(* Logix 5000 project; controller LeakTestAuto vendor 1 type 14 code 226 rev 37.11; software revision 37.01; part 9 of 12 *)
(* tags used below, declared in another part *)
   AOI_Barcode_Comms : AOI_CommStatus;
   AOI_CTS1_Comms : AOI_CommStatus;
   AOI_CTS2_Comms : AOI_CommStatus;
   AOI_RFID_Comms : AOI_CommStatus;
   AOI_RFID_LoadingNest_Comms : AOI_CommStatus;
   AOI_Robot_Comms : AOI_CommStatus;
   BarcodeScanner : udt_OutputStructure;
   Conveyor : udt_OutputStructure;
   Conveyor_Seq : udt_SequenceStructure_X64;
   ConveyorCleatSensorFault : BOOL;
   FailCount : COUNTER;
   HMI_OP220_ClearProcessFaultCounts_IND : BOOL;
   HMI_OP220_ClearProcessFaultCounts_PB : BOOL;
   LastFaults : DINT[2];
   LeakTester1 : udt_OutputStructure;
   LeakTester2 : udt_OutputStructure;
   Nest1Cylinder : udt_OutputStructure;
   Nest2Cylinder : udt_OutputStructure;
   OP220 : udt_Mode;
   OP220_Disable3510 : BOOL;
   OP220_Fault_Counter : COUNTER;
   OP220_Fault_Counter_ONS : BOOL;
   OP220_Fault_Number : DINT;
   OP220_Fault_Reset_ONS : BOOL;
   OP220_FaultCounter_Reset_ONS : BOOL;
   OP220_LeakTest : udt_ProcessFault;
   OP220_ProcessFaultsONS : DINT;
   OP220_Seq : udt_SequenceStructure_X64;
   RFID_Comp : AOI_RFIDCompare;
   RFID_DiagData : DINT[4];
   RFID_ExpectedFixtureVal : SINT[5,12];
   RFID_LoadingNestDiagData : DINT[4];
   RFID_LoadingNestReceiveBuffer : SINT[8000];
   RFID_LoadingNestSendBuffer : SINT[8000];
   RFID_PortOffset : DINT;
   RFID_ReceiveBuffer : SINT[8000];
   RFID_RWHAllPort : RWH_CMD;
   RFID_RWHLoadingNest : RWH_CMD;
   RFID_SendBuffer : SINT[8000];
   RFID_TagStatus : BOOL[32];
   RFIDLoadingNestScanner : udt_OutputStructure;
   RFIDScanner : udt_OutputStructure;
   Robot : udt_OutputStructure;
   RobotGripper : udt_OutputStructure;
   RobotInputs : udt_EpsonInputs;
   TON_Cylinder1DownTimeout : TIMER;
   TON_Cylinder1UpTimeout : TIMER;
   TON_Cylinder2DownTimeout : TIMER;
   TON_Cylinder2UpTimeout : TIMER;
   TON_FailChute : TIMER[10];
   TON_Nest2CylinderTimer : TIMER;
   I_OP220_N3_MAIN_AIR_OK : ALIAS FOR Local:3:I.Pt07.Data;
   I_OP220_N3_NEST2_EXTEND : ALIAS FOR Local:3:I.Pt06.Data;
   I_OP220_N3_NEST2_HOME : ALIAS FOR Local:3:I.Pt05.Data;
   I_OP220_N3_REJECT_BIN_OK : ALIAS FOR Local:3:I.Pt09.Data;
   I_OP220_N4_DC_OK : ALIAS FOR Local:4:I.Pt01.Data;
   I_OP220_N4_DC_OK_PS2 : ALIAS FOR Local:4:I.Pt04.Data;
   James_Dint : DINT;   // James Test Word
   O_OP220_N5_EN_NEST2_EXT : ALIAS FOR Local:5:O.Pt07.Data;
   O_OP220_N5_EN_NEST2_HOME : ALIAS FOR Local:5:O.Pt08.Data;
   OP220_ConsumedFromMain : DINT[50];
   OP220_EStopTest_DCS : DCI_STOP;
   PLC : AOI_PLC;
   ShiftChange : BOOL;
(* MainProgram, continued *)

ROUTINE R61_Nest2Cylinder   (* ladder *)
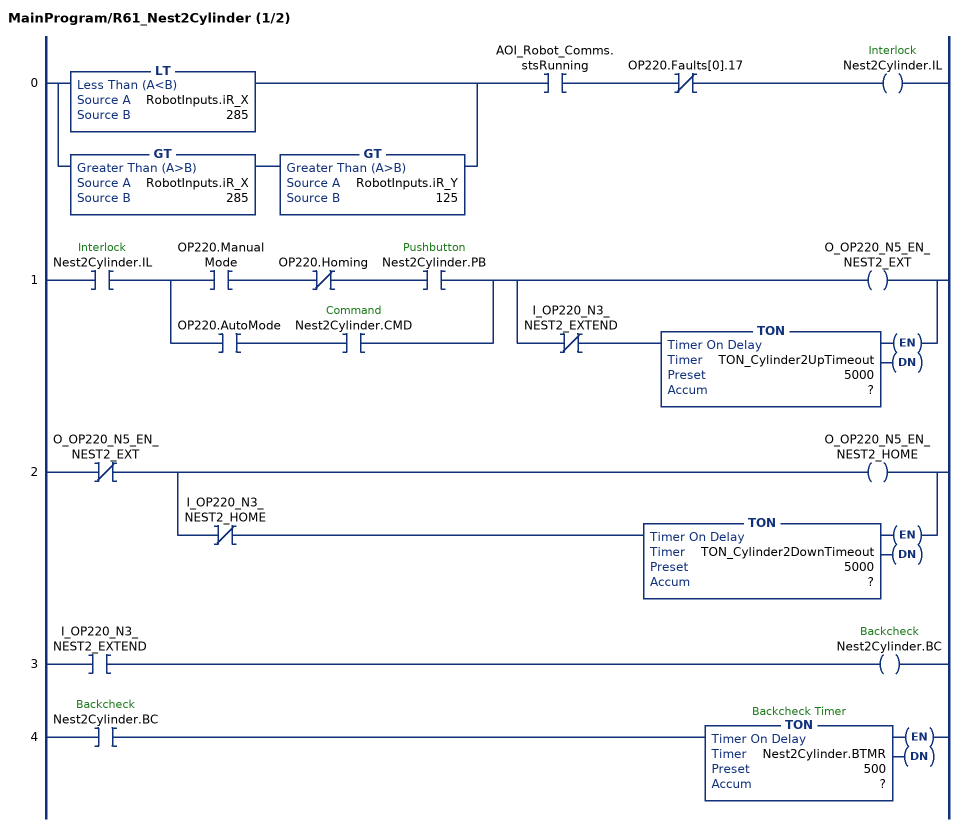
   0: [LT(RobotInputs.iR_X,285) ,GT(RobotInputs.iR_X,285) GT(RobotInputs.iR_Y,125) ]XIC(AOI_Robot_Comms.stsRunning)XIO(OP220.Faults[0].17)OTE(Nest2Cylinder.IL);
   1: XIC(Nest2Cylinder.IL)[XIC(OP220.ManualMode) XIO(OP220.Homing) XIC(Nest2Cylinder.PB) ,XIC(OP220.AutoMode) XIC(Nest2Cylinder.CMD) ][OTE(O_OP220_N5_EN_NEST2_EXT) ,XIO(I_OP220_N3_NEST2_EXTEND) TON(TON_Cylinder2UpTimeout,?,?) ];
   2: XIO(O_OP220_N5_EN_NEST2_EXT)[OTE(O_OP220_N5_EN_NEST2_HOME) ,XIO(I_OP220_N3_NEST2_HOME) TON(TON_Cylinder2DownTimeout,?,?) ];
   3: XIC(I_OP220_N3_NEST2_EXTEND)OTE(Nest2Cylinder.BC);
   4: XIC(Nest2Cylinder.BC)TON(Nest2Cylinder.BTMR,?,?);
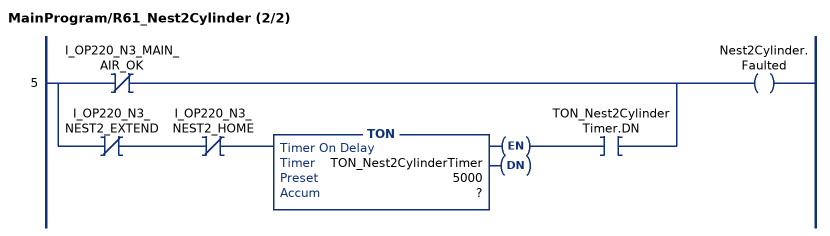
   5: [XIO(I_OP220_N3_MAIN_AIR_OK) ,XIO(I_OP220_N3_NEST2_EXTEND) XIO(I_OP220_N3_NEST2_HOME) TON(TON_Nest2CylinderTimer,?,?) XIC(TON_Nest2CylinderTimer.DN) ]OTE(Nest2Cylinder.Faulted);
END_ROUTINE

ROUTINE R70_RFID   (* ladder *)
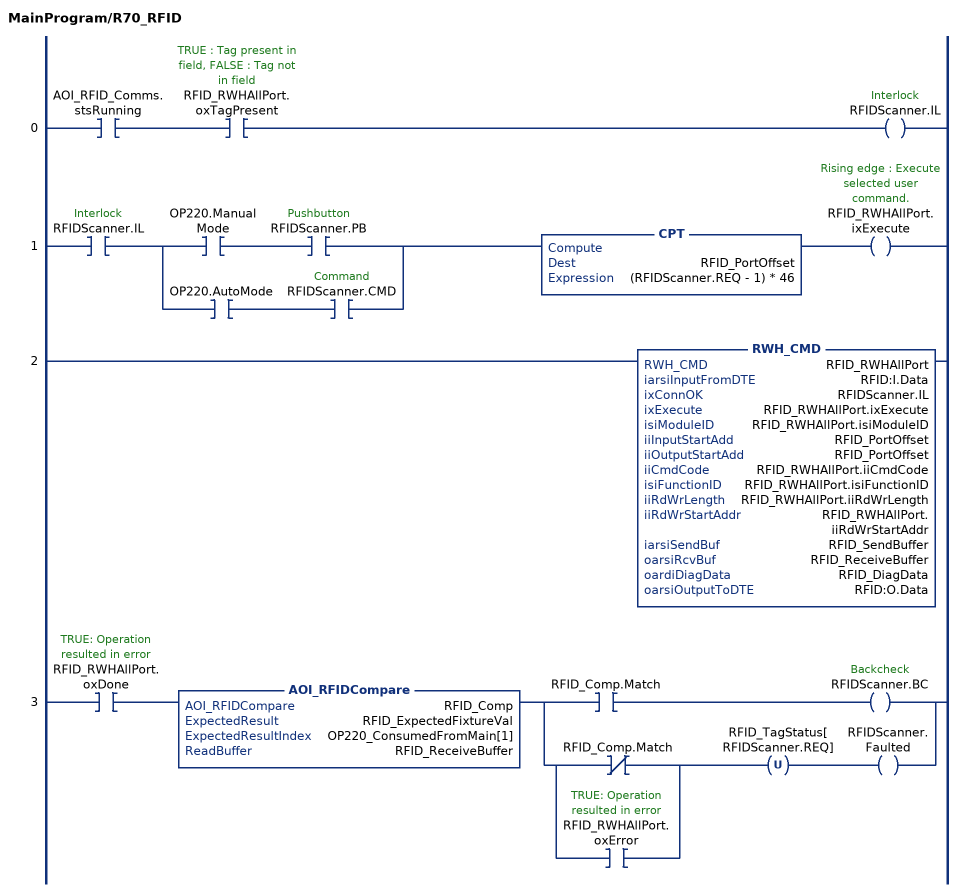
   0: XIC(AOI_RFID_Comms.stsRunning)XIC(RFID_RWHAllPort.oxTagPresent)OTE(RFIDScanner.IL);
   1: XIC(RFIDScanner.IL)[XIC(OP220.ManualMode) XIC(RFIDScanner.PB) ,XIC(OP220.AutoMode) XIC(RFIDScanner.CMD) ]CPT(RFID_PortOffset,(RFIDScanner.REQ - 1) * 46)OTE(RFID_RWHAllPort.ixExecute);
   2: RWH_CMD(RFID_RWHAllPort,RFID:I.Data,RFIDScanner.IL,RFID_RWHAllPort.ixExecute,RFID_RWHAllPort.isiModuleID,RFID_PortOffset,RFID_PortOffset,RFID_RWHAllPort.iiCmdCode,RFID_RWHAllPort.isiFunctionID,RFID_RWHAllPort.iiRdWrLength,RFID_RWHAllPort.iiRdWrStartAddr,RFID_SendBuffer,RFID_ReceiveBuffer,RFID_DiagData,RFID:O.Data);
   3: XIC(RFID_RWHAllPort.oxDone)AOI_RFIDCompare(RFID_Comp,RFID_ExpectedFixtureVal,OP220_ConsumedFromMain[1],RFID_ReceiveBuffer)[XIC(RFID_Comp.Match) OTE(RFIDScanner.BC) ,[XIO(RFID_Comp.Match) ,XIC(RFID_RWHAllPort.oxError) ] OTU(RFID_TagStatus[RFIDScanner.REQ]) OTE(RFIDScanner.Faulted) ];
END_ROUTINE

ROUTINE R71_RFID_LoadingNest   (* ladder *)
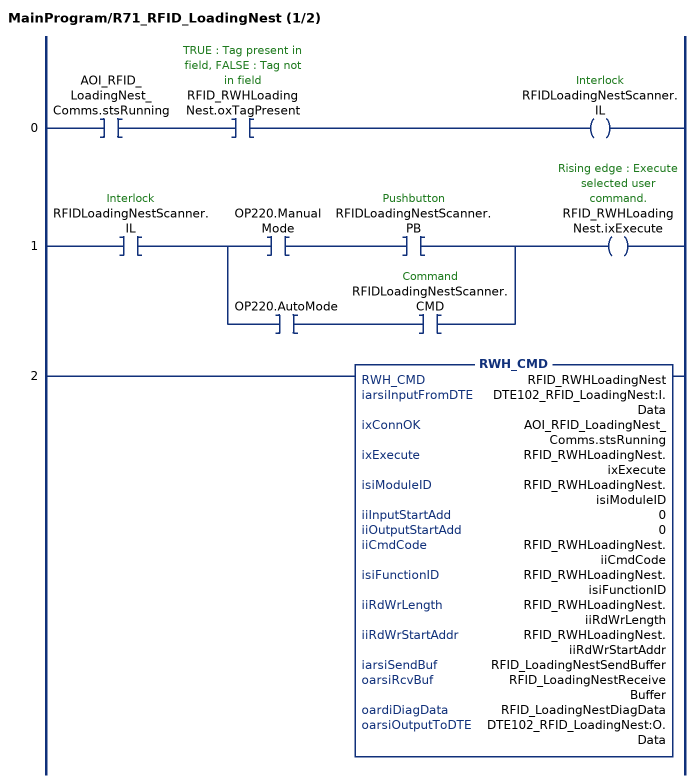
   0: XIC(AOI_RFID_LoadingNest_Comms.stsRunning)XIC(RFID_RWHLoadingNest.oxTagPresent)OTE(RFIDLoadingNestScanner.IL);
   1: XIC(RFIDLoadingNestScanner.IL)[XIC(OP220.ManualMode) XIC(RFIDLoadingNestScanner.PB) ,XIC(OP220.AutoMode) XIC(RFIDLoadingNestScanner.CMD) ]OTE(RFID_RWHLoadingNest.ixExecute);
   2: RWH_CMD(RFID_RWHLoadingNest,DTE102_RFID_LoadingNest:I.Data,AOI_RFID_LoadingNest_Comms.stsRunning,RFID_RWHLoadingNest.ixExecute,RFID_RWHLoadingNest.isiModuleID,0,0,RFID_RWHLoadingNest.iiCmdCode,RFID_RWHLoadingNest.isiFunctionID,RFID_RWHLoadingNest.iiRdWrLength,RFID_RWHLoadingNest.iiRdWrStartAddr,RFID_LoadingNestSendBuffer,RFID_LoadingNestReceiveBuffer,RFID_LoadingNestDiagData,DTE102_RFID_LoadingNest:O.Data);
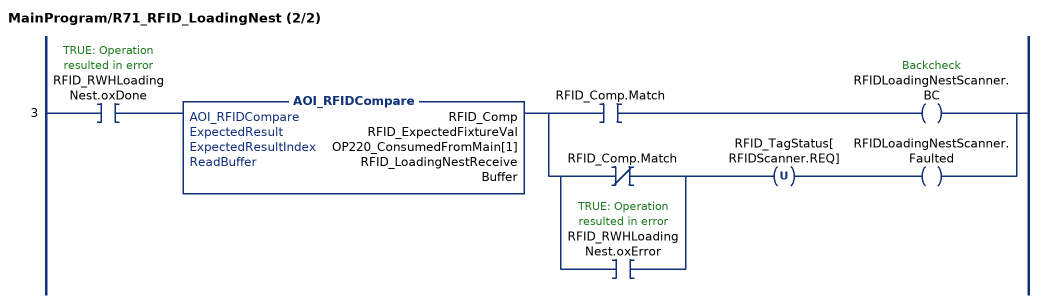
   3: XIC(RFID_RWHLoadingNest.oxDone)AOI_RFIDCompare(RFID_Comp,RFID_ExpectedFixtureVal,OP220_ConsumedFromMain[1],RFID_LoadingNestReceiveBuffer)[XIC(RFID_Comp.Match) OTE(RFIDLoadingNestScanner.BC) ,[XIO(RFID_Comp.Match) ,XIC(RFID_RWHLoadingNest.oxError) ] OTU(RFID_TagStatus[RFIDScanner.REQ]) OTE(RFIDLoadingNestScanner.Faulted) ];
END_ROUTINE

ROUTINE R89_3_5_10_Alarms   (* ladder *)
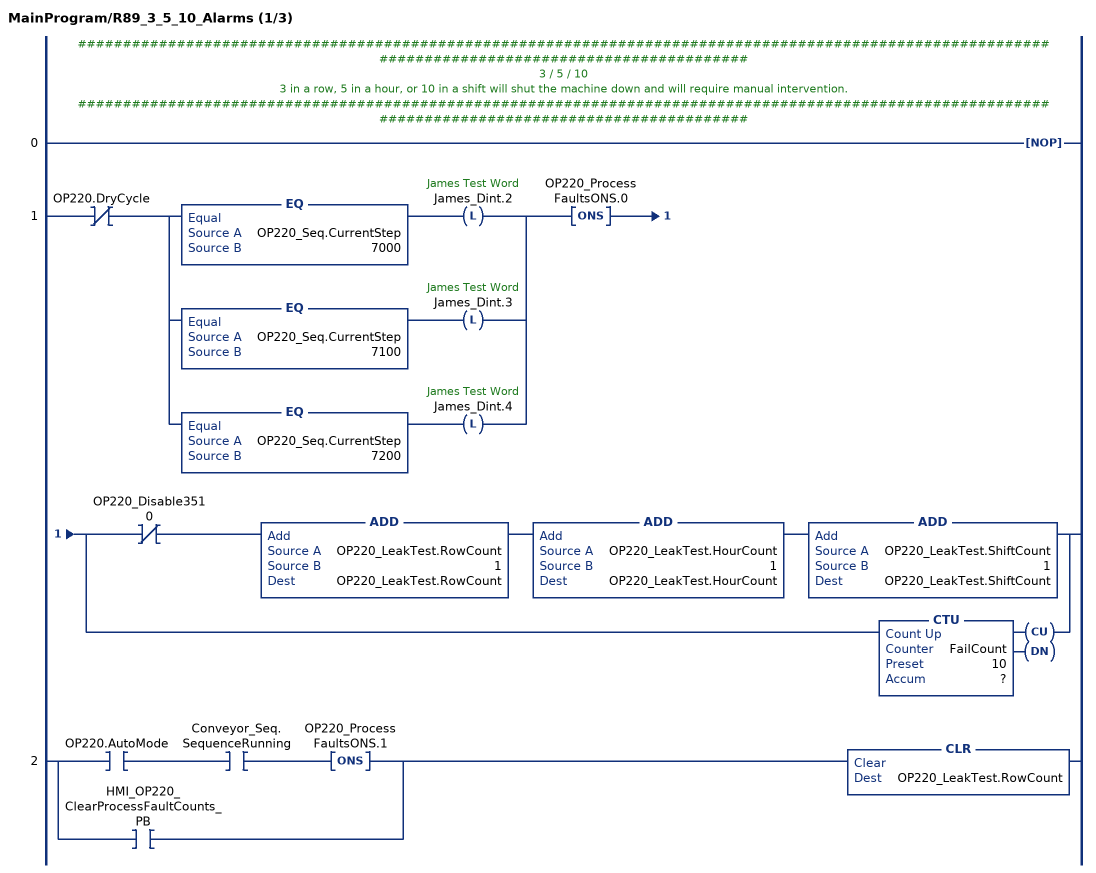
   // #####################################################################################################################################################
   // 3 / 5 / 10
   // 	3 in a row, 5 in a hour, or 10 in a shift will shut the machine down and will require manual intervention.
   // #####################################################################################################################################################
   0: NOP();
   1: XIO(OP220.DryCycle)[EQ(OP220_Seq.CurrentStep,7000) OTL(James_Dint.2) ,EQ(OP220_Seq.CurrentStep,7100) OTL(James_Dint.3) ,EQ(OP220_Seq.CurrentStep,7200) OTL(James_Dint.4) ]ONS(OP220_ProcessFaultsONS.0)[XIO(OP220_Disable3510) ADD(OP220_LeakTest.RowCount,1,OP220_LeakTest.RowCount) ADD(OP220_LeakTest.HourCount,1,OP220_LeakTest.HourCount) ADD(OP220_LeakTest.ShiftCount,1,OP220_LeakTest.ShiftCount) ,CTU(FailCount,?,?) ];
   2: [XIC(OP220.AutoMode) XIC(Conveyor_Seq.SequenceRunning) ONS(OP220_ProcessFaultsONS.1) ,XIC(HMI_OP220_ClearProcessFaultCounts_PB) ]CLR(OP220_LeakTest.RowCount);
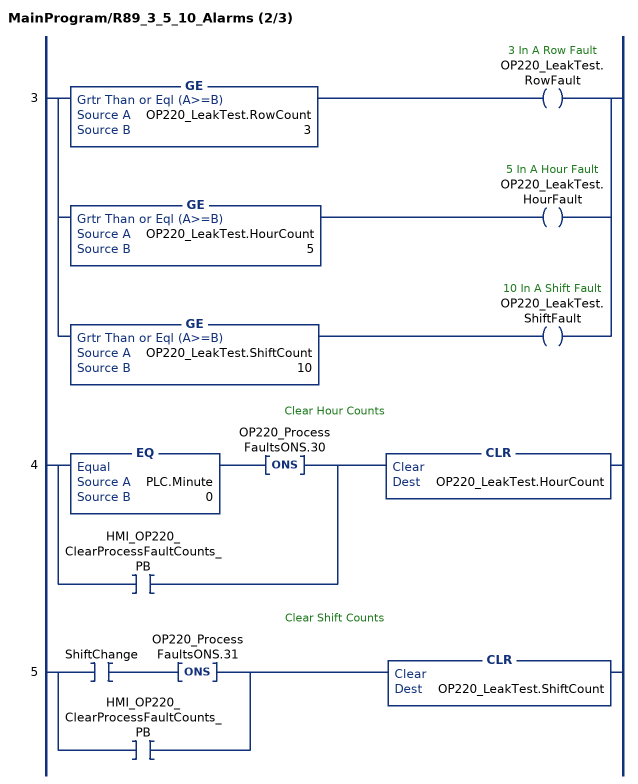
   3: [GE(OP220_LeakTest.RowCount,3) OTE(OP220_LeakTest.RowFault) ,GE(OP220_LeakTest.HourCount,5) OTE(OP220_LeakTest.HourFault) ,GE(OP220_LeakTest.ShiftCount,10) OTE(OP220_LeakTest.ShiftFault) ];
   // Clear Hour Counts
   4: [EQ(PLC.Minute,0) ONS(OP220_ProcessFaultsONS.30) ,XIC(HMI_OP220_ClearProcessFaultCounts_PB) ]CLR(OP220_LeakTest.HourCount);
   // Clear Shift Counts
   5: [XIC(ShiftChange) ONS(OP220_ProcessFaultsONS.31) ,XIC(HMI_OP220_ClearProcessFaultCounts_PB) ]CLR(OP220_LeakTest.ShiftCount);
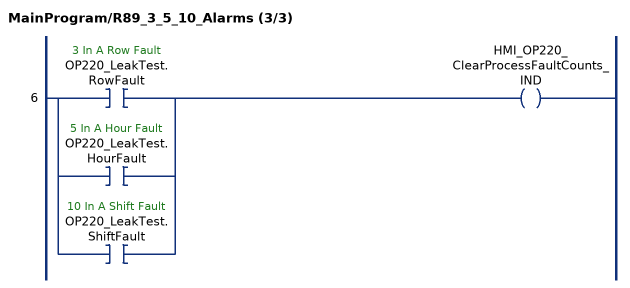
   6: [XIC(OP220_LeakTest.RowFault) ,XIC(OP220_LeakTest.HourFault) ,XIC(OP220_LeakTest.ShiftFault) ]OTE(HMI_OP220_ClearProcessFaultCounts_IND);
END_ROUTINE

ROUTINE R90_Faults   (* ladder *)
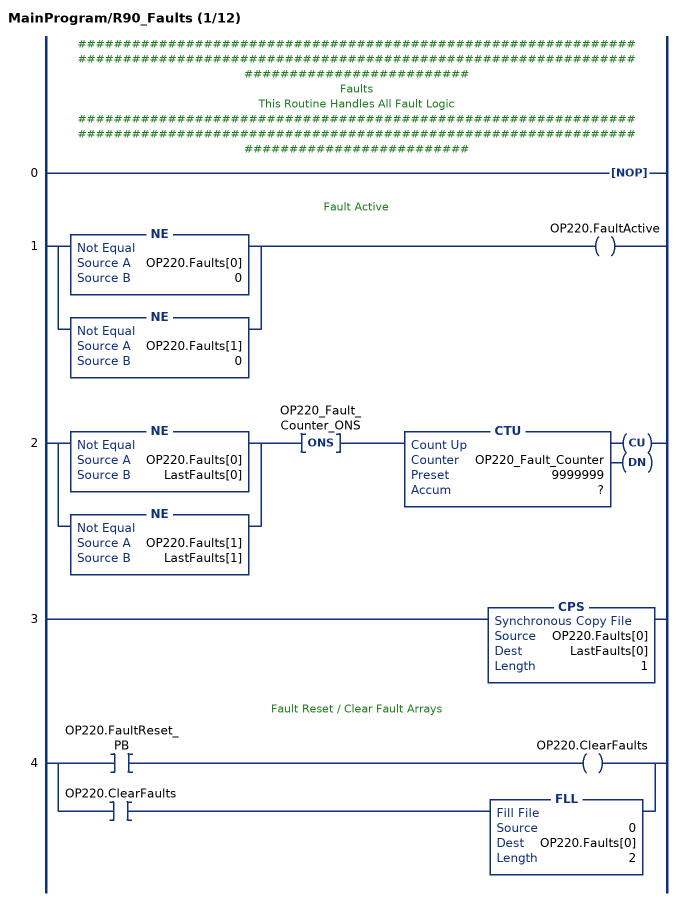
   // #####################################################################################################################################################
   // Faults
   // This Routine Handles All Fault Logic
   // #####################################################################################################################################################
   0: NOP();
   // Fault Active
   1: [NE(OP220.Faults[0],0) ,NE(OP220.Faults[1],0) ]OTE(OP220.FaultActive);
   2: [NE(OP220.Faults[0],LastFaults[0]) ,NE(OP220.Faults[1],LastFaults[1]) ]ONS(OP220_Fault_Counter_ONS)CTU(OP220_Fault_Counter,?,?);
   3: CPS(OP220.Faults[0],LastFaults[0],1);
   // Fault Reset / Clear Fault Arrays
   4: [XIC(OP220.FaultReset_PB) OTE(OP220.ClearFaults) ,XIC(OP220.ClearFaults) FLL(0,OP220.Faults[0],2) ];
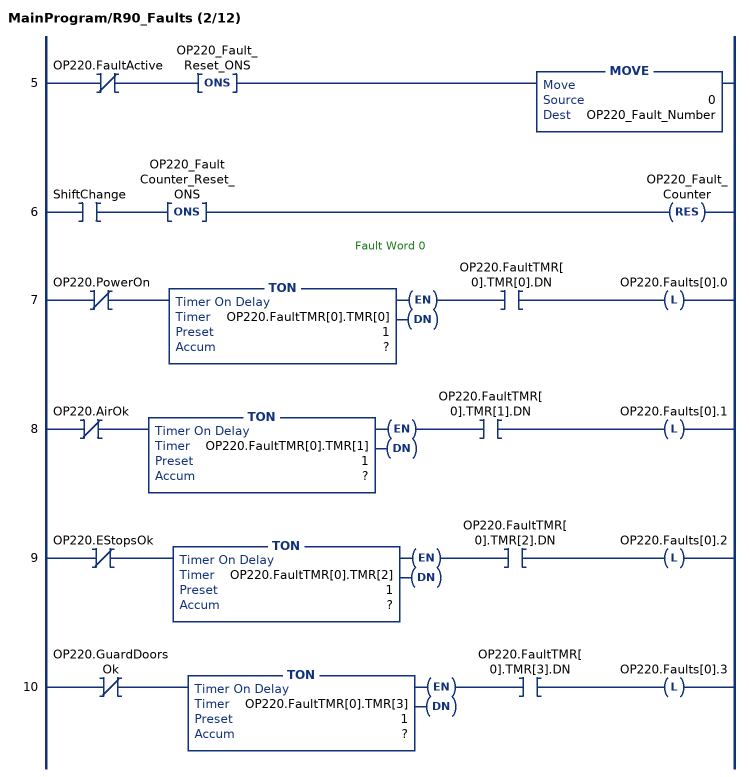
   5: XIO(OP220.FaultActive)ONS(OP220_Fault_Reset_ONS)MOVE(0,OP220_Fault_Number);
   6: XIC(ShiftChange)ONS(OP220_FaultCounter_Reset_ONS)RES(OP220_Fault_Counter);
   // Fault Word 0
   7: XIO(OP220.PowerOn)TON(OP220.FaultTMR[0].TMR[0],?,?)XIC(OP220.FaultTMR[0].TMR[0].DN)OTL(OP220.Faults[0].0);
   8: XIO(OP220.AirOk)TON(OP220.FaultTMR[0].TMR[1],?,?)XIC(OP220.FaultTMR[0].TMR[1].DN)OTL(OP220.Faults[0].1);
   9: XIO(OP220.EStopsOk)TON(OP220.FaultTMR[0].TMR[2],?,?)XIC(OP220.FaultTMR[0].TMR[2].DN)OTL(OP220.Faults[0].2);
   10: XIO(OP220.GuardDoorsOk)TON(OP220.FaultTMR[0].TMR[3],?,?)XIC(OP220.FaultTMR[0].TMR[3].DN)OTL(OP220.Faults[0].3);
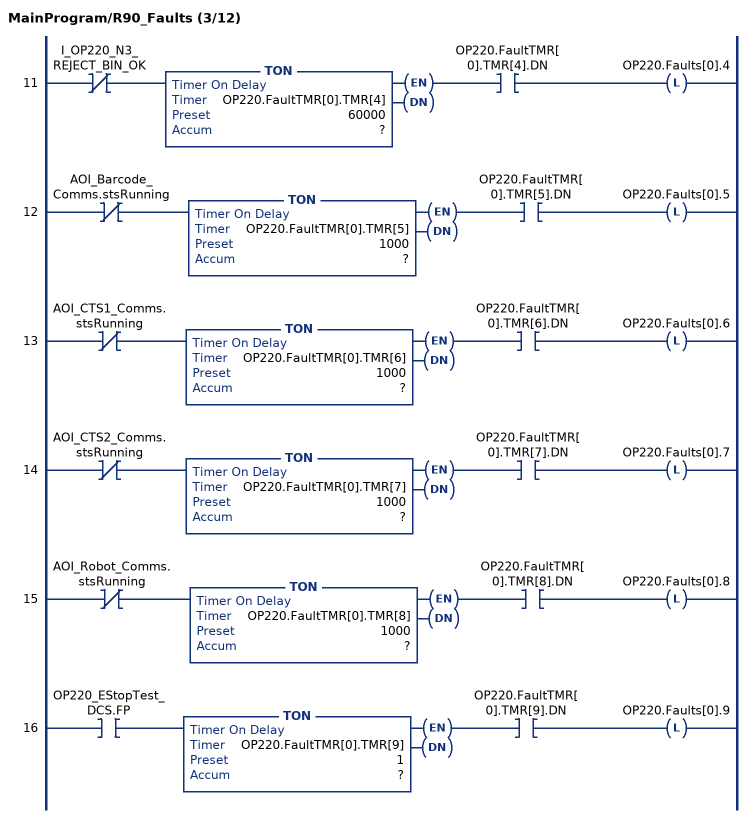
   11: XIO(I_OP220_N3_REJECT_BIN_OK)TON(OP220.FaultTMR[0].TMR[4],?,?)XIC(OP220.FaultTMR[0].TMR[4].DN)OTL(OP220.Faults[0].4);
   12: XIO(AOI_Barcode_Comms.stsRunning)TON(OP220.FaultTMR[0].TMR[5],?,?)XIC(OP220.FaultTMR[0].TMR[5].DN)OTL(OP220.Faults[0].5);
   13: XIO(AOI_CTS1_Comms.stsRunning)TON(OP220.FaultTMR[0].TMR[6],?,?)XIC(OP220.FaultTMR[0].TMR[6].DN)OTL(OP220.Faults[0].6);
   14: XIO(AOI_CTS2_Comms.stsRunning)TON(OP220.FaultTMR[0].TMR[7],?,?)XIC(OP220.FaultTMR[0].TMR[7].DN)OTL(OP220.Faults[0].7);
   15: XIO(AOI_Robot_Comms.stsRunning)TON(OP220.FaultTMR[0].TMR[8],?,?)XIC(OP220.FaultTMR[0].TMR[8].DN)OTL(OP220.Faults[0].8);
   16: XIC(OP220_EStopTest_DCS.FP)TON(OP220.FaultTMR[0].TMR[9],?,?)XIC(OP220.FaultTMR[0].TMR[9].DN)OTL(OP220.Faults[0].9);
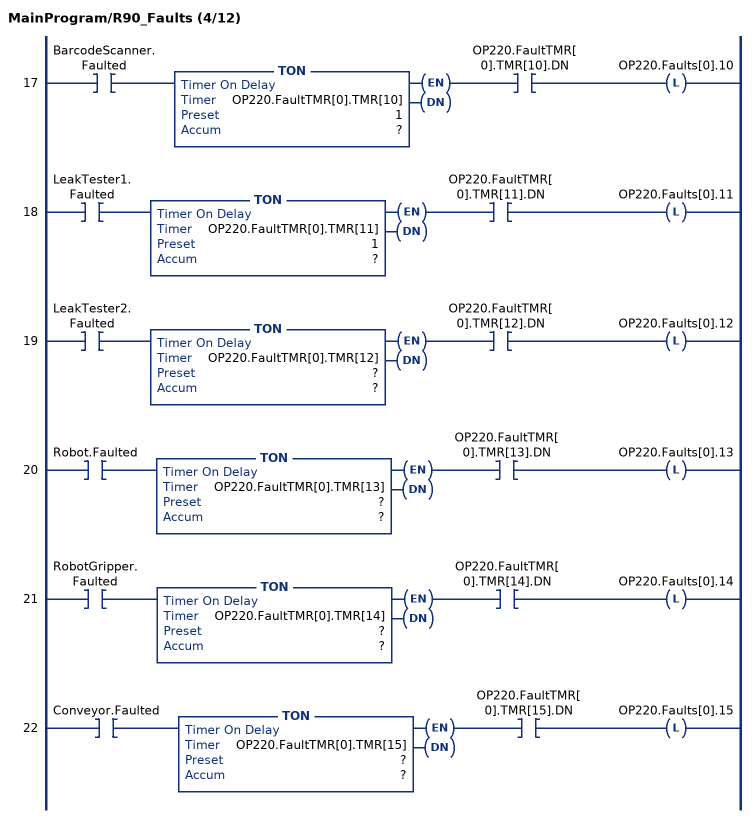
   17: XIC(BarcodeScanner.Faulted)TON(OP220.FaultTMR[0].TMR[10],?,?)XIC(OP220.FaultTMR[0].TMR[10].DN)OTL(OP220.Faults[0].10);
   18: XIC(LeakTester1.Faulted)TON(OP220.FaultTMR[0].TMR[11],?,?)XIC(OP220.FaultTMR[0].TMR[11].DN)OTL(OP220.Faults[0].11);
   19: XIC(LeakTester2.Faulted)TON(OP220.FaultTMR[0].TMR[12],?,?)XIC(OP220.FaultTMR[0].TMR[12].DN)OTL(OP220.Faults[0].12);
   20: XIC(Robot.Faulted)TON(OP220.FaultTMR[0].TMR[13],?,?)XIC(OP220.FaultTMR[0].TMR[13].DN)OTL(OP220.Faults[0].13);
   21: XIC(RobotGripper.Faulted)TON(OP220.FaultTMR[0].TMR[14],?,?)XIC(OP220.FaultTMR[0].TMR[14].DN)OTL(OP220.Faults[0].14);
   22: XIC(Conveyor.Faulted)TON(OP220.FaultTMR[0].TMR[15],?,?)XIC(OP220.FaultTMR[0].TMR[15].DN)OTL(OP220.Faults[0].15);
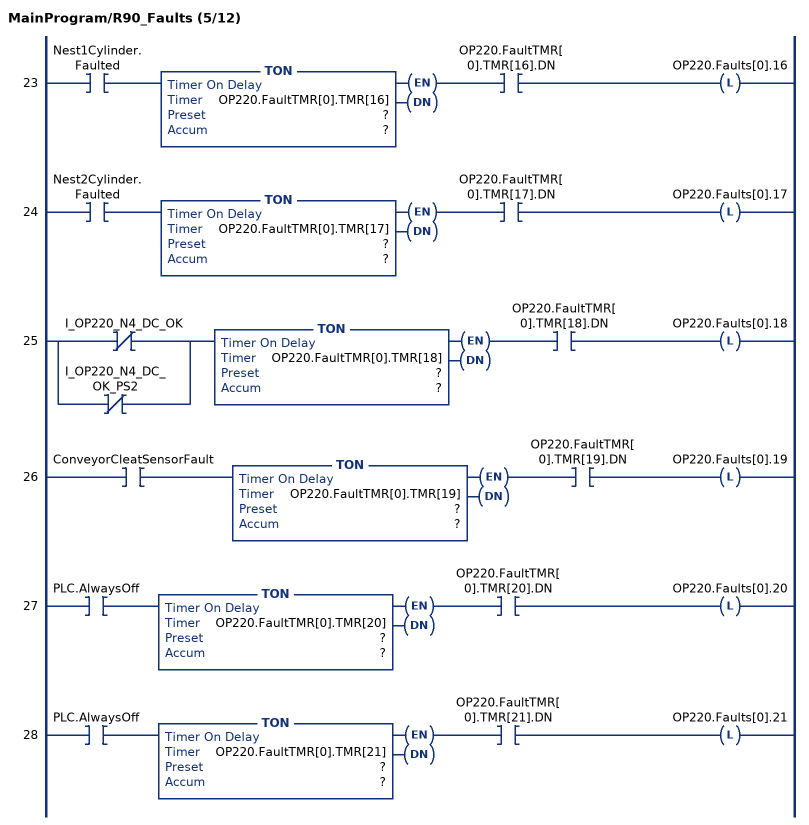
   23: XIC(Nest1Cylinder.Faulted)TON(OP220.FaultTMR[0].TMR[16],?,?)XIC(OP220.FaultTMR[0].TMR[16].DN)OTL(OP220.Faults[0].16);
   24: XIC(Nest2Cylinder.Faulted)TON(OP220.FaultTMR[0].TMR[17],?,?)XIC(OP220.FaultTMR[0].TMR[17].DN)OTL(OP220.Faults[0].17);
   25: [XIO(I_OP220_N4_DC_OK) ,XIO(I_OP220_N4_DC_OK_PS2) ]TON(OP220.FaultTMR[0].TMR[18],?,?)XIC(OP220.FaultTMR[0].TMR[18].DN)OTL(OP220.Faults[0].18);
   26: XIC(ConveyorCleatSensorFault)TON(OP220.FaultTMR[0].TMR[19],?,?)XIC(OP220.FaultTMR[0].TMR[19].DN)OTL(OP220.Faults[0].19);
   27: XIC(PLC.AlwaysOff)TON(OP220.FaultTMR[0].TMR[20],?,?)XIC(OP220.FaultTMR[0].TMR[20].DN)OTL(OP220.Faults[0].20);
   28: XIC(PLC.AlwaysOff)TON(OP220.FaultTMR[0].TMR[21],?,?)XIC(OP220.FaultTMR[0].TMR[21].DN)OTL(OP220.Faults[0].21);
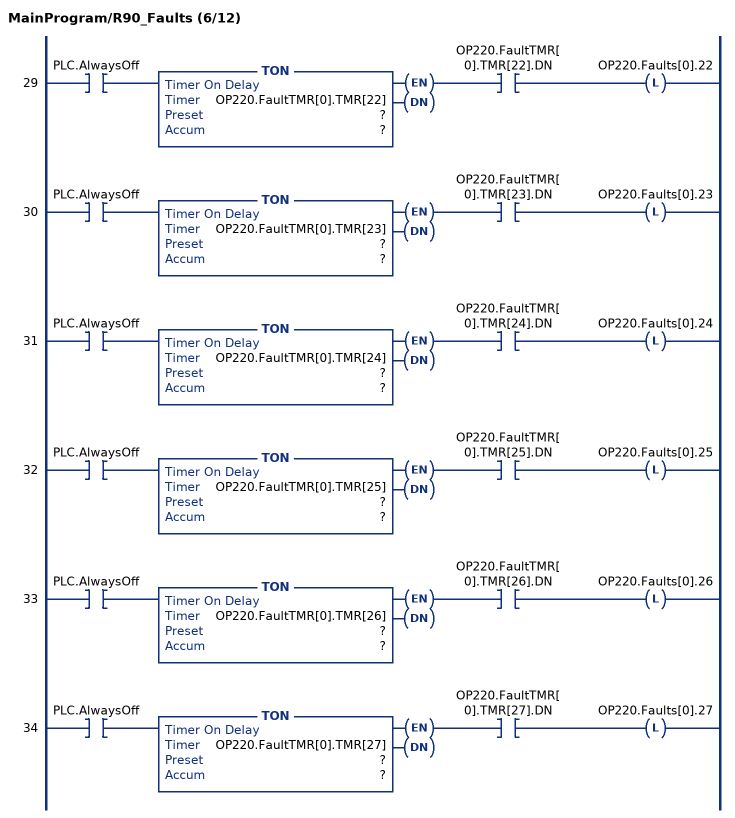
   29: XIC(PLC.AlwaysOff)TON(OP220.FaultTMR[0].TMR[22],?,?)XIC(OP220.FaultTMR[0].TMR[22].DN)OTL(OP220.Faults[0].22);
   30: XIC(PLC.AlwaysOff)TON(OP220.FaultTMR[0].TMR[23],?,?)XIC(OP220.FaultTMR[0].TMR[23].DN)OTL(OP220.Faults[0].23);
   31: XIC(PLC.AlwaysOff)TON(OP220.FaultTMR[0].TMR[24],?,?)XIC(OP220.FaultTMR[0].TMR[24].DN)OTL(OP220.Faults[0].24);
   32: XIC(PLC.AlwaysOff)TON(OP220.FaultTMR[0].TMR[25],?,?)XIC(OP220.FaultTMR[0].TMR[25].DN)OTL(OP220.Faults[0].25);
   33: XIC(PLC.AlwaysOff)TON(OP220.FaultTMR[0].TMR[26],?,?)XIC(OP220.FaultTMR[0].TMR[26].DN)OTL(OP220.Faults[0].26);
   34: XIC(PLC.AlwaysOff)TON(OP220.FaultTMR[0].TMR[27],?,?)XIC(OP220.FaultTMR[0].TMR[27].DN)OTL(OP220.Faults[0].27);
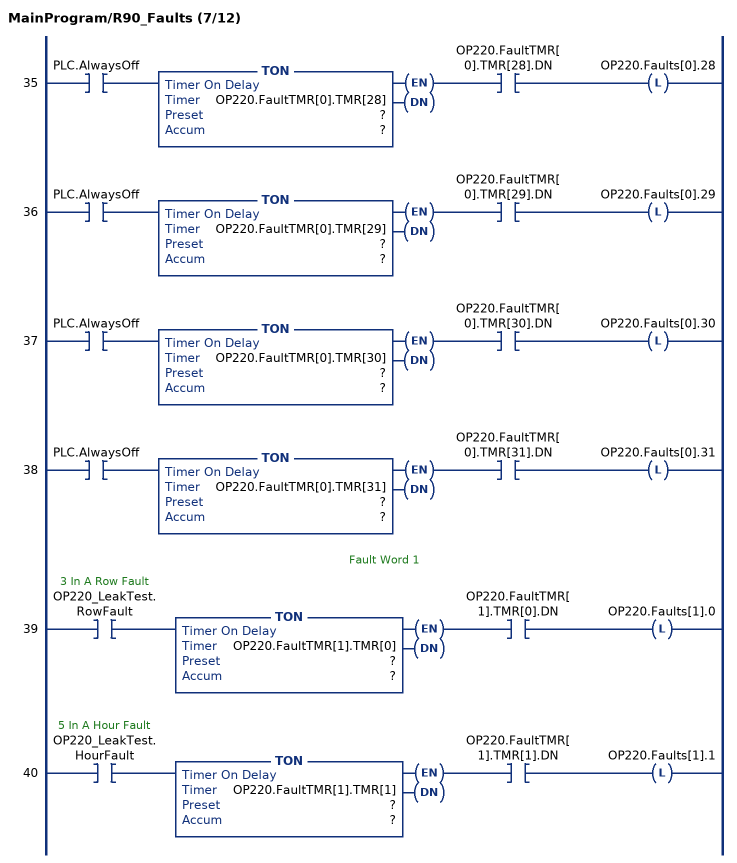
   35: XIC(PLC.AlwaysOff)TON(OP220.FaultTMR[0].TMR[28],?,?)XIC(OP220.FaultTMR[0].TMR[28].DN)OTL(OP220.Faults[0].28);
   36: XIC(PLC.AlwaysOff)TON(OP220.FaultTMR[0].TMR[29],?,?)XIC(OP220.FaultTMR[0].TMR[29].DN)OTL(OP220.Faults[0].29);
   37: XIC(PLC.AlwaysOff)TON(OP220.FaultTMR[0].TMR[30],?,?)XIC(OP220.FaultTMR[0].TMR[30].DN)OTL(OP220.Faults[0].30);
   38: XIC(PLC.AlwaysOff)TON(OP220.FaultTMR[0].TMR[31],?,?)XIC(OP220.FaultTMR[0].TMR[31].DN)OTL(OP220.Faults[0].31);
   // Fault Word 1
   39: XIC(OP220_LeakTest.RowFault)TON(OP220.FaultTMR[1].TMR[0],?,?)XIC(OP220.FaultTMR[1].TMR[0].DN)OTL(OP220.Faults[1].0);
   40: XIC(OP220_LeakTest.HourFault)TON(OP220.FaultTMR[1].TMR[1],?,?)XIC(OP220.FaultTMR[1].TMR[1].DN)OTL(OP220.Faults[1].1);
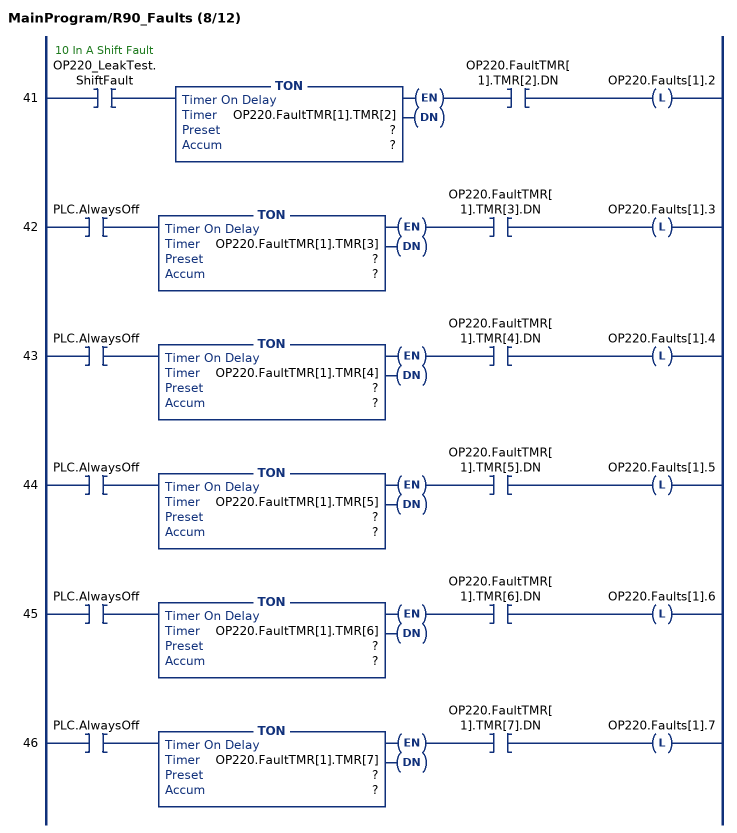
   41: XIC(OP220_LeakTest.ShiftFault)TON(OP220.FaultTMR[1].TMR[2],?,?)XIC(OP220.FaultTMR[1].TMR[2].DN)OTL(OP220.Faults[1].2);
   42: XIC(PLC.AlwaysOff)TON(OP220.FaultTMR[1].TMR[3],?,?)XIC(OP220.FaultTMR[1].TMR[3].DN)OTL(OP220.Faults[1].3);
   43: XIC(PLC.AlwaysOff)TON(OP220.FaultTMR[1].TMR[4],?,?)XIC(OP220.FaultTMR[1].TMR[4].DN)OTL(OP220.Faults[1].4);
   44: XIC(PLC.AlwaysOff)TON(OP220.FaultTMR[1].TMR[5],?,?)XIC(OP220.FaultTMR[1].TMR[5].DN)OTL(OP220.Faults[1].5);
   45: XIC(PLC.AlwaysOff)TON(OP220.FaultTMR[1].TMR[6],?,?)XIC(OP220.FaultTMR[1].TMR[6].DN)OTL(OP220.Faults[1].6);
   46: XIC(PLC.AlwaysOff)TON(OP220.FaultTMR[1].TMR[7],?,?)XIC(OP220.FaultTMR[1].TMR[7].DN)OTL(OP220.Faults[1].7);
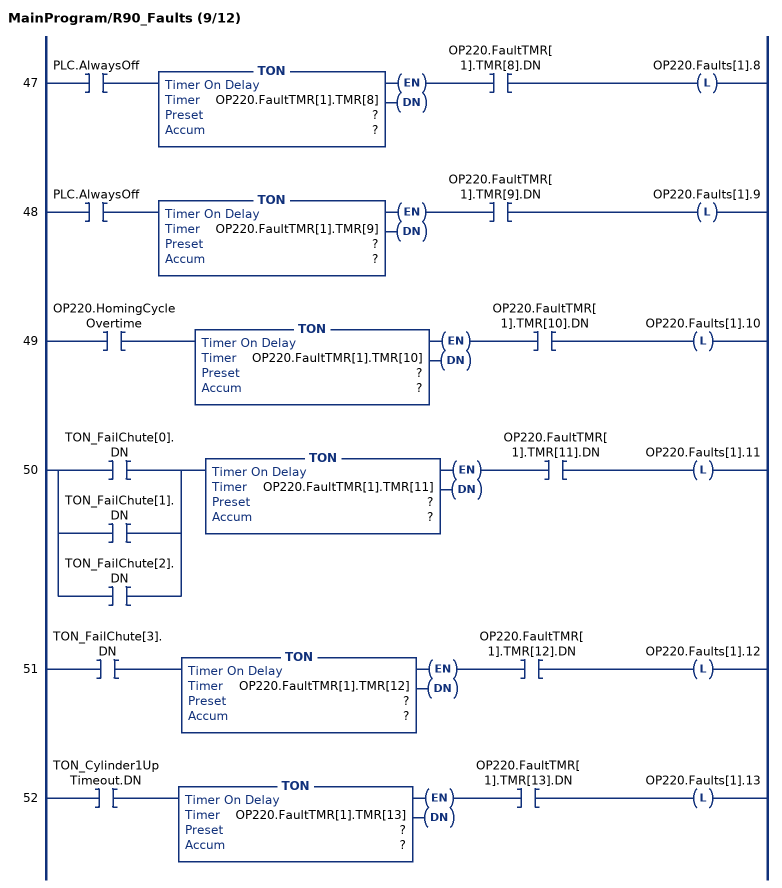
   47: XIC(PLC.AlwaysOff)TON(OP220.FaultTMR[1].TMR[8],?,?)XIC(OP220.FaultTMR[1].TMR[8].DN)OTL(OP220.Faults[1].8);
   48: XIC(PLC.AlwaysOff)TON(OP220.FaultTMR[1].TMR[9],?,?)XIC(OP220.FaultTMR[1].TMR[9].DN)OTL(OP220.Faults[1].9);
   49: XIC(OP220.HomingCycleOvertime)TON(OP220.FaultTMR[1].TMR[10],?,?)XIC(OP220.FaultTMR[1].TMR[10].DN)OTL(OP220.Faults[1].10);
   50: [XIC(TON_FailChute[0].DN) ,XIC(TON_FailChute[1].DN) ,XIC(TON_FailChute[2].DN) ]TON(OP220.FaultTMR[1].TMR[11],?,?)XIC(OP220.FaultTMR[1].TMR[11].DN)OTL(OP220.Faults[1].11);
   51: XIC(TON_FailChute[3].DN)TON(OP220.FaultTMR[1].TMR[12],?,?)XIC(OP220.FaultTMR[1].TMR[12].DN)OTL(OP220.Faults[1].12);
   52: XIC(TON_Cylinder1UpTimeout.DN)TON(OP220.FaultTMR[1].TMR[13],?,?)XIC(OP220.FaultTMR[1].TMR[13].DN)OTL(OP220.Faults[1].13);
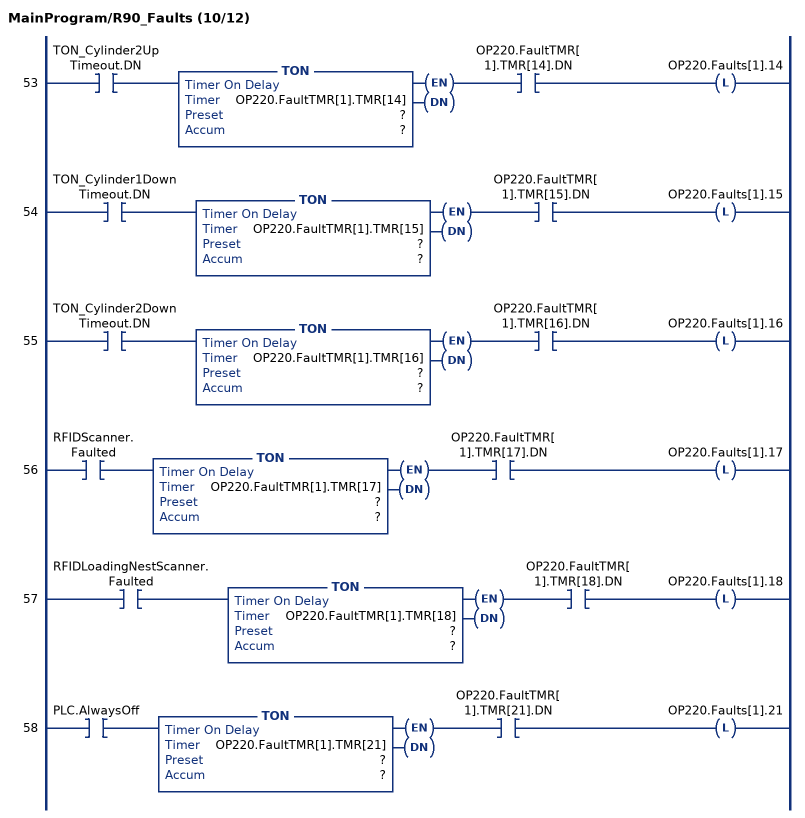
   53: XIC(TON_Cylinder2UpTimeout.DN)TON(OP220.FaultTMR[1].TMR[14],?,?)XIC(OP220.FaultTMR[1].TMR[14].DN)OTL(OP220.Faults[1].14);
   54: XIC(TON_Cylinder1DownTimeout.DN)TON(OP220.FaultTMR[1].TMR[15],?,?)XIC(OP220.FaultTMR[1].TMR[15].DN)OTL(OP220.Faults[1].15);
   55: XIC(TON_Cylinder2DownTimeout.DN)TON(OP220.FaultTMR[1].TMR[16],?,?)XIC(OP220.FaultTMR[1].TMR[16].DN)OTL(OP220.Faults[1].16);
   56: XIC(RFIDScanner.Faulted)TON(OP220.FaultTMR[1].TMR[17],?,?)XIC(OP220.FaultTMR[1].TMR[17].DN)OTL(OP220.Faults[1].17);
   57: XIC(RFIDLoadingNestScanner.Faulted)TON(OP220.FaultTMR[1].TMR[18],?,?)XIC(OP220.FaultTMR[1].TMR[18].DN)OTL(OP220.Faults[1].18);
   58: XIC(PLC.AlwaysOff)TON(OP220.FaultTMR[1].TMR[21],?,?)XIC(OP220.FaultTMR[1].TMR[21].DN)OTL(OP220.Faults[1].21);
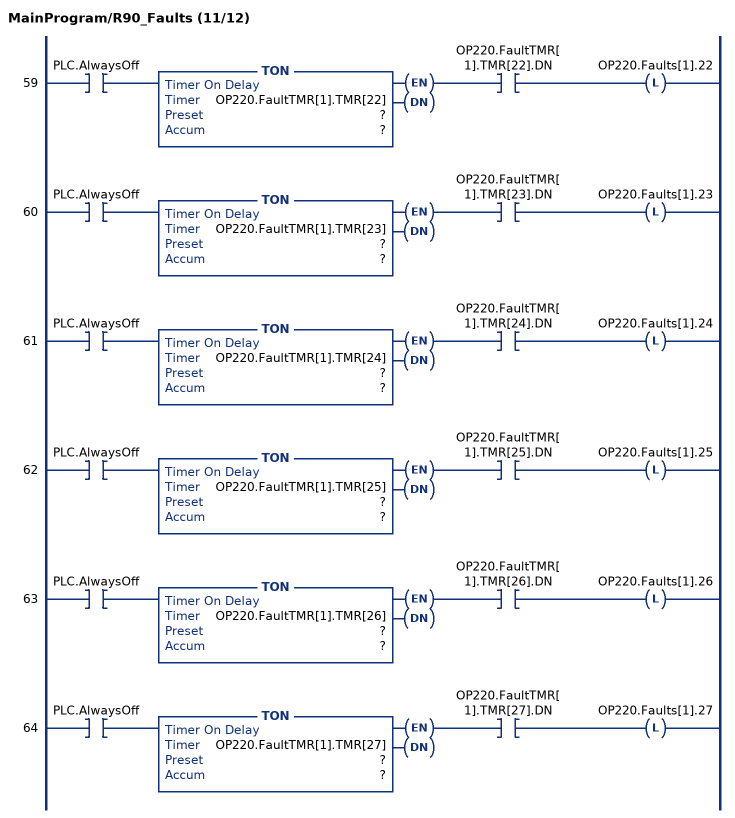
   59: XIC(PLC.AlwaysOff)TON(OP220.FaultTMR[1].TMR[22],?,?)XIC(OP220.FaultTMR[1].TMR[22].DN)OTL(OP220.Faults[1].22);
   60: XIC(PLC.AlwaysOff)TON(OP220.FaultTMR[1].TMR[23],?,?)XIC(OP220.FaultTMR[1].TMR[23].DN)OTL(OP220.Faults[1].23);
   61: XIC(PLC.AlwaysOff)TON(OP220.FaultTMR[1].TMR[24],?,?)XIC(OP220.FaultTMR[1].TMR[24].DN)OTL(OP220.Faults[1].24);
   62: XIC(PLC.AlwaysOff)TON(OP220.FaultTMR[1].TMR[25],?,?)XIC(OP220.FaultTMR[1].TMR[25].DN)OTL(OP220.Faults[1].25);
   63: XIC(PLC.AlwaysOff)TON(OP220.FaultTMR[1].TMR[26],?,?)XIC(OP220.FaultTMR[1].TMR[26].DN)OTL(OP220.Faults[1].26);
   64: XIC(PLC.AlwaysOff)TON(OP220.FaultTMR[1].TMR[27],?,?)XIC(OP220.FaultTMR[1].TMR[27].DN)OTL(OP220.Faults[1].27);
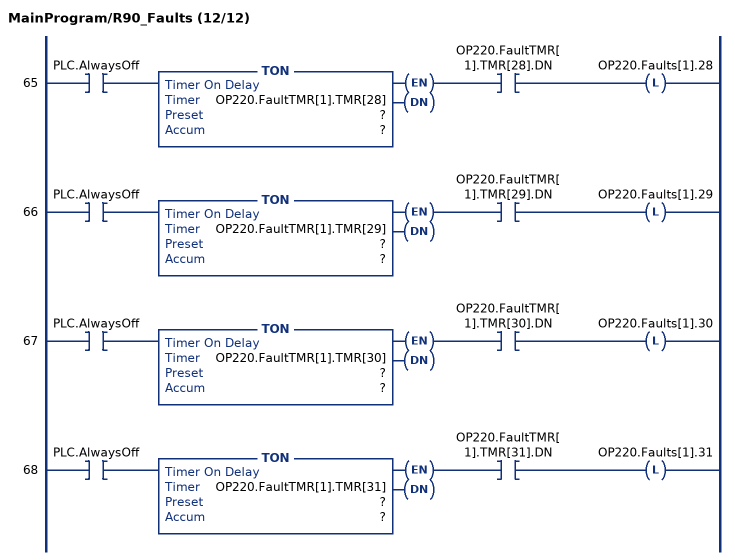
   65: XIC(PLC.AlwaysOff)TON(OP220.FaultTMR[1].TMR[28],?,?)XIC(OP220.FaultTMR[1].TMR[28].DN)OTL(OP220.Faults[1].28);
   66: XIC(PLC.AlwaysOff)TON(OP220.FaultTMR[1].TMR[29],?,?)XIC(OP220.FaultTMR[1].TMR[29].DN)OTL(OP220.Faults[1].29);
   67: XIC(PLC.AlwaysOff)TON(OP220.FaultTMR[1].TMR[30],?,?)XIC(OP220.FaultTMR[1].TMR[30].DN)OTL(OP220.Faults[1].30);
   68: XIC(PLC.AlwaysOff)TON(OP220.FaultTMR[1].TMR[31],?,?)XIC(OP220.FaultTMR[1].TMR[31].DN)OTL(OP220.Faults[1].31);
END_ROUTINE
